(*
An interface which can be implemented by various event storage function blocks.
*)

INTERFACE i_Persistent_Event_Storage

METHOD Store_Event
VAR_INPUT
	st_Event_To_Store : st_Event;
END_VAR
END_METHOD

END_INTERFACE

(* stored: Version 1.1.0.1
   Itf i_Persistent_Event_Storage: Id {17fa3198-a6f3-48ab-b464-70345ab51de4}
   Method Store_Event: Id {ecd44b3e-378f-4a8c-ba36-10e08db7dc86} *)
